PROGRAM WX_CP_Simple
VAR
	WX1A_Clamp : SimpleClamp;
	WX1B_Clamp : SimpleClamp;
	
	WX2A_Clamp : SimpleClamp;
	WX2B_Clamp : SimpleClamp;
	
	WX3A_Clamp : SimpleClamp;
	WX3B_Clamp : SimpleClamp;
	
	WX4A_Clamp : SimpleClamp;
	WX4B_Clamp : SimpleClamp;
END_VAR

//WX1
WX1B_Clamp(Limit_NC_NO_CI := 0);
WX1A_Clamp(Limit_NC_NO_CI := 0);

//WX2
WX2A_Clamp(Limit_NC_NO_CI := 0);
WX2B_Clamp(Limit_NC_NO_CI := 0);

//WX3
WX3A_Clamp(Limit_NC_NO_CI := 0);
WX3B_Clamp(Limit_NC_NO_CI := 0);

//WX4
WX4A_Clamp(Limit_NC_NO_CI := 0);
WX4B_Clamp(Limit_NC_NO_CI := 0);

END_PROGRAM

(* stored: Version 1.1.0.1, ProductVersion 3.1.4024.12
   POU WX_CP_Simple: Id {b343d1dc-837f-4a71-8ef3-3d0cc6e5233f}, SpecialFunc None *)
